FUNCTION proj1_TupleStruct_1: LREAL
{ S7_Optimized_Access := 'true' }
    VAR_INPUT
        tuple: TupleStruct_1;
    END_VAR

BEGIN
    proj1_TupleStruct_1 := tuple.field1;
END_FUNCTION
